PROGRAM Receitas
VAR
	AUX_FS				:BOOL := FALSE;	//Auxiliar do First Scan
	FS					:BOOL;			//First Scan
	iCounter			:INT;			//Contador para o FOR
	IndiceReceita		:INT;			//Índice da receita que está na interface
	NomeReceita			:STRING:='SELECIONAR RECEITA';	//Nome da receita selecionada
	IndiceReceitaAtiva	:INT;			//Índice da receita ativa
	
	Teste:INT;/////////////////////////////////////////
	
	//Comandos
	Salvar				:BOOL;	//Salva a receita na memória
	Excluir				:BOOL;	//Exclui a receita selecionada
	Atualizar			:BOOL;	//É executado quando a receita do ComboBox é trocada. Ele atualiza os dados da tela com a receita selecionada
	CarregarReceita		:BOOL;	//Envia a receita de interface para a máquina
	NomeExistente		:BOOL;	//Se verdadeiro, o nome escolhido já está em uso
	ReceitaOK			:BOOL;	//Receita com todos os parâmetros preenchidos corretamente
	ReceitaCarregada	:BOOL;	//Carrega para a interface a receita que está carregada na máquina
	i					:INT;	// Variável para iteração do FOR
	TempoAux			:REAL;	//Variável auxiliar para cálculo de tempo da receita
	TempoDosPassos		:ARRAY[1..12] OF DINT;	//Esse array salva, no índice dos passos, o tempo do mesmo. No final, tudo é somado para retornar o tempo da batelada
	TempoTotal			:DINT;	//Tempo total da receita
END_VAR

// FS é um pulso do primeiro scan do CLP
FS := NOT AUX_FS;
aux_fs := TRUE;

Receta_Activa.interfaceSetNombreRecetaActiva := SEL(IndiceReceita > 0, '', RecetasGestion.BibliotecaRecetas[IndiceReceita].Nombre);

// No primeiro scan do CLP, os ID's das receitas são configurados e se o texto delas estiver vazio, é setado para "Vazio"
//Cada ID deve ser único para que o Combobox funcione corretamente

IF FS THEN
	LiqNaReceita();
	FOR iCounter := 1 TO 100 BY 1 DO
  		RecetasGestion.aComboboxRecipes[iCounter].id := iCounter;
		IF RecetasGestion.aComboboxRecipes[iCounter].text = '' THEN
			RecetasGestion.aComboboxRecipes[iCounter].text := 'Vazio';
		END_IF;
	END_FOR;
	
END_IF;

//Salva a receita que foi editada
IF Salvar THEN
	FOR iCounter := 1 TO 100 DO	//A receita salva não pode ter o mesmo nome de outra já salva
		IF NomeReceita = RecetasGestion.BibliotecaRecetas[iCounter].Nombre AND  IndiceReceita <> iCounter AND NomeReceita <> '' THEN	//A receita selecionada pode continuar com o mesmo nome
			NomeExistente := TRUE;
			EXIT;
		END_IF
	END_FOR
	IF NomeReceita <> '' AND NOT NomeExistente THEN
		RecetasGestion.BibliotecaRecetas[IndiceReceita].Nombre				:= NomeReceita;
		RecetasGestion.aComboboxRecipes[IndiceReceita].text					:= NomeReceita;
		RecetasGestion.BibliotecaRecetas[IndiceReceita].SetTmrDescarga		:= Receta_Activa.interfaceSetTmrDescarga;
		RecetasGestion.BibliotecaRecetas[IndiceReceita].SetTmrHomogenizado	:= Receta_Activa.interfaceSetTmrHomogenizado;
		RecetasGestion.BibliotecaRecetas[IndiceReceita].SetVelocDescarga	:= Receta_Activa.interfaceSetVelocDescarga;
		RecetasGestion.BibliotecaRecetas[IndiceReceita].SetVelocHomogenizado := Receta_Activa.interfaceSetVelocHomogenizado;
		RecetasGestion.BibliotecaRecetas[IndiceReceita].SetCircuitosLiq		:= Receta_Activa.interfaceSetCircuitosLiq;
		RecetasGestion.BibliotecaRecetas[IndiceReceita].SetCircuitosPo		:= Receta_Activa.interfaceSetCircuitosPo;
		RecetasGestion.BibliotecaRecetas[IndiceReceita].Aspiracao			:= Receta_Activa.interfaceSetAspiracao;
		
		NomeReceita := Receta_Activa.interfaceSetNombreRecetaActiva;
	END_IF;
		
	Salvar := FALSE;
END_IF

//É executado quando a receita do ComboBox é trocada. Ele atualiza os dados da tela com a receita selecionada
IF Atualizar THEN
	IF IndiceReceita = 0 THEN
		IndiceReceita := 1;
	END_IF
	LiqNaReceita();
	
	NomeReceita := RecetasGestion.BibliotecaRecetas[IndiceReceita].Nombre;
	Receta_Activa.interfaceSetTmrDescarga		:= RecetasGestion.BibliotecaRecetas[IndiceReceita].SetTmrDescarga;
	Receta_Activa.interfaceSetTmrHomogenizado	:= RecetasGestion.BibliotecaRecetas[IndiceReceita].SetTmrHomogenizado;
	Receta_Activa.interfaceSetVelocDescarga		:= RecetasGestion.BibliotecaRecetas[IndiceReceita].SetVelocDescarga;
	Receta_Activa.interfaceSetVelocHomogenizado	:= RecetasGestion.BibliotecaRecetas[IndiceReceita].SetVelocHomogenizado;
	Receta_Activa.interfaceSetCircuitosLiq		:= RecetasGestion.BibliotecaRecetas[IndiceReceita].SetCircuitosLiq;
	Receta_Activa.interfaceSetCircuitosPo		:= RecetasGestion.BibliotecaRecetas[IndiceReceita].SetCircuitosPo;
	Receta_Activa.interfaceSetAspiracao			:= RecetasGestion.BibliotecaRecetas[IndiceReceita].Aspiracao;
	//Receta_Activa.interfaceSetTiempoTotal		:= RecetasGestion.BibliotecaRecetas[IndiceReceita].SetTiempoTotal;
	Atualizar := FALSE;
END_IF

//Esse bloco exclui os dados de uma receita salva
IF Excluir THEN
		RecetasGestion.BibliotecaRecetas[IndiceReceita].Nombre := '';
		RecetasGestion.aComboboxRecipes[IndiceReceita].text := 'Vazio';
		RecetasGestion.BibliotecaRecetas[IndiceReceita].SetTmrDescarga := 0;
		RecetasGestion.BibliotecaRecetas[IndiceReceita].SetTmrHomogenizado := 0;
		RecetasGestion.BibliotecaRecetas[IndiceReceita].SetVelocDescarga := 0;
		RecetasGestion.BibliotecaRecetas[IndiceReceita].SetVelocHomogenizado := 0;
		RecetasGestion.BibliotecaRecetas[IndiceReceita].Aspiracao := FALSE;
		Receta_Activa.SetNombreRecetaActiva := '';
		Receta_Activa.interfaceSetAspiracao := FALSE;
		
		FOR iCounter := 1 TO 12 BY 1 DO
			RecetasGestion.BibliotecaRecetas[IndiceReceita].SetCircuitosLiq[iCounter].Demora	:= 0;
			RecetasGestion.BibliotecaRecetas[IndiceReceita].SetCircuitosLiq[iCounter].Dosis		:= 0;
			RecetasGestion.BibliotecaRecetas[IndiceReceita].SetCircuitosLiq[iCounter].Inyeccion	:= 0;
			RecetasGestion.BibliotecaRecetas[IndiceReceita].SetCircuitosLiq[iCounter].Paso		:= 0;
		END_FOR
		FOR iCounter := 1 TO 4 BY 1 DO
			RecetasGestion.BibliotecaRecetas[IndiceReceita].SetCircuitosPo[iCounter].Demora		:= 0;
			RecetasGestion.BibliotecaRecetas[IndiceReceita].SetCircuitosPo[iCounter].Dosis		:= 0;
			RecetasGestion.BibliotecaRecetas[IndiceReceita].SetCircuitosPo[iCounter].Inyeccion	:= 0;
			RecetasGestion.BibliotecaRecetas[IndiceReceita].SetCircuitosPo[iCounter].Paso		:= 0;
		END_FOR
		Excluir := FALSE;
END_IF

//Carrega a receita que está sendo editada para a máquina
IF CarregarReceita THEN
	Receta_Activa.SetNombreRecetaActiva	:= RecetasGestion.BibliotecaRecetas[IndiceReceita].Nombre;
	Receta_Activa.SetTmrHomogenizado	:= Receta_Activa.interfaceSetTmrHomogenizado;
	Receta_Activa.SetTmrDescarga		:= Receta_Activa.interfaceSetTmrDescarga;
	Receta_Activa.SetVelocHomogenizado	:= Receta_Activa.interfaceSetVelocHomogenizado;
	Receta_Activa.SetVelocDescarga		:= Receta_Activa.interfaceSetVelocDescarga;
	Receta_Activa.SetCircuitosLiq		:= Receta_Activa.interfaceSetCircuitosLiq;
	Receta_Activa.SetCircuitosPo		:= Receta_Activa.interfaceSetCircuitosPo;
	Receta_Activa.SetTiempoTotal		:= Receta_Activa.interfaceSetTiempoTotal;
	Receta_Activa.SetAspiracao		:= Receta_Activa.interfaceSetAspiracao;
	CarregarReceita := FALSE;
	LiqNaReceita();
END_IF

//Verificação se a receita pode ser salva/carregada. 
//A receita não pode ser carregada/salva se não houver nenhum líquido/pó ou se houver algum com os parametros de dosagem zerado
ReceitaOK := TRUE;

//Verifica se tem algum líquido colocado na sequência
FOR iCounter :=  1 TO 12 BY 1 DO
	IF Receta_Activa.interfaceSetCircuitosLiq[iCounter].Paso <> 0 THEN
		ReceitaOK := TRUE;
		EXIT;
	ELSE
		Teste := 100 + iCounter;
		ReceitaOK := FALSE;
	END_IF
END_FOR


//Verifica se os liquidos na sequencia estão com a dosagem preenchida
IF ReceitaOK THEN
	FOR iCounter :=  1 TO 12 BY 1 DO
		IF Receta_Activa.interfaceSetCircuitosLiq[iCounter].Paso <> 0 THEN
			IF Receta_Activa.interfaceSetCircuitosLiq[iCounter].Dosis <= 0 OR Receta_Activa.interfaceSetCircuitosLiq[iCounter].Inyeccion <= 0 THEN
				ReceitaOK := FALSE;
				Teste := 200 + iCounter;
				EXIT;
			END_IF;
		END_IF;	
	END_FOR
END_IF

//Verifica se tem pó na receita
FOR iCounter :=  1 TO 4 BY 1 DO
	IF Receta_Activa.InterfaceSetCircuitosPo[iCounter].Paso <> 0 THEN
		IF Receta_Activa.InterfaceSetCircuitosPo[iCounter].Dosis <= 0 OR Receta_Activa.InterfaceSetCircuitosPo[iCounter].Inyeccion <= 0 THEN
			ReceitaOK := FALSE;
			EXIT;
		END_IF;
	END_IF
END_FOR


//Cálculo do tempo da receita
FOR i := 1 TO 12 DO
	TempoDosPassos[i] := 0;
END_FOR
TempoAux := 0;
FOR i := 1 TO 12 DO
	//Verifica os tempos dos líquidos
	IF TempoAux = 0 OR Receta_Activa.interfaceSetCircuitosLiq[i].Demora + Receta_Activa.interfaceSetCircuitosLiq[i].Inyeccion > TempoAux THEN
		TempoAux := Receta_Activa.interfaceSetCircuitosLiq[i].Demora + Receta_Activa.interfaceSetCircuitosLiq[i].Inyeccion;
		IF Receta_Activa.interfaceSetCircuitosLiq[i].Paso > 0 THEN
			IF TO_DINT(TempoAux) > TempoDosPassos[Receta_Activa.interfaceSetCircuitosLiq[i].Paso] THEN
				TempoDosPassos[Receta_Activa.interfaceSetCircuitosLiq[i].Paso] := TO_DINT(TempoAux);
			END_IF
		END_IF
	END_IF
	TempoAux := 0;
END_FOR

FOR i := 1 TO 12 DO
	IF Receta_Activa.interfaceSetCircuitosPo[1].Paso = i THEN
		IF Receta_Activa.interfaceSetCircuitosPo[1].Demora + Receta_Activa.interfaceSetCircuitosPo[1].Inyeccion > TempoDosPassos[i] THEN
			TempoDosPassos[i] := Receta_Activa.interfaceSetCircuitosPo[1].Demora + Receta_Activa.interfaceSetCircuitosPo[1].Inyeccion;
		END_IF
	END_IF
	IF Receta_Activa.interfaceSetCircuitosPo[2].Paso = i THEN
		IF Receta_Activa.interfaceSetCircuitosPo[2].Demora + Receta_Activa.interfaceSetCircuitosPo[2].Inyeccion > TempoDosPassos[i] THEN
			TempoDosPassos[i] := Receta_Activa.interfaceSetCircuitosPo[2].Demora + Receta_Activa.interfaceSetCircuitosPo[2].Inyeccion;
		END_IF
	END_IF
END_FOR

TempoTotal := 0;
FOR i := 1 TO 12 DO
	TempoTotal := TempoTotal + TempoDosPassos[i];
END_FOR

TempoTotal := TempoTotal + Receta_Activa.interfaceSetTmrDescarga + Receta_Activa.interfaceSetTmrHomogenizado;
Receta_Activa.interfaceSetTiempoTotal := TO_REAL(TempoTotal);


//Lógica do botão "CARREGADA". Serve para que o operador carregue para a interface a receita que está na máquina.
IF ReceitaCarregada THEN
	FOR i := 1 TO 100 DO
		IF RecetasGestion.aComboboxRecipes[i].text = Receta_Activa.SetNombreRecetaActiva THEN
			IndiceReceita := RecetasGestion.aComboboxRecipes[i].id;
			EXIT;
		END_IF
	END_FOR
	//Receta_Activa.interfaceSetNombreRecetaActiva := CONCAT(Receta_Activa.interfaceSetNombreRecetaActiva, TO_STRING(" - EM PROCESSO"));
	Receta_Activa.interfaceSetCircuitosLiq		:= Receta_Activa.SetCircuitosLiq;
	Receta_Activa.interfaceSetCircuitosPo		:= Receta_Activa.SetCircuitosPo;
	Receta_Activa.interfaceSetNombreRecetaActiva	:= Receta_Activa.SetNombreRecetaActiva;
	Receta_Activa.interfaceSetTiempoTotal		:= Receta_Activa.SetTiempoTotal;
	Receta_Activa.interfaceSetTmrDescarga		:= Receta_Activa.SetTmrDescarga;
	Receta_Activa.interfaceSetTmrHomogenizado	:= Receta_Activa.SetTmrHomogenizado;
	Receta_Activa.interfaceSetVelocDescarga		:= Receta_Activa.SetVelocDescarga;
	Receta_Activa.interfaceSetVelocHomogenizado	:= Receta_Activa.SetVelocDescarga;
	Receta_Activa.interfaceSetAspiracao			:= Receta_Activa.SetAspiracao;
	ReceitaCarregada := FALSE;
END_IF

END_PROGRAM

(* stored: Version 1.1.0.1, ProductVersion 3.1.4024.14
   POU Receitas: Id {a811645b-e664-4b28-b8de-1aab1d692da5}, SpecialFunc None *)
